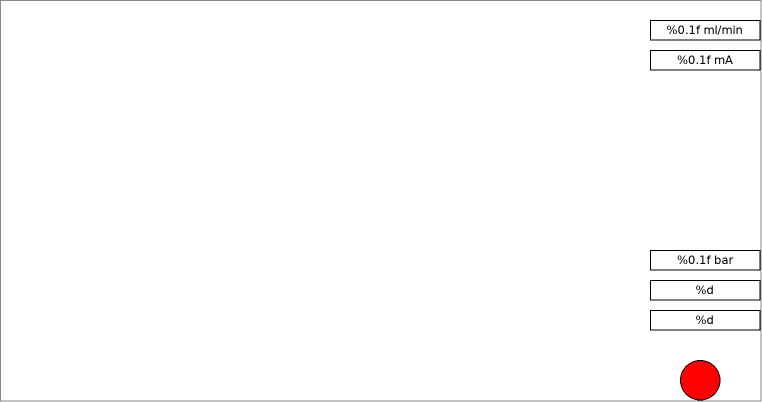
VISUALIZATION Q1  // 762x402
    Rectangle (650,20 110x20), "%0.1f ml/min", text variable: IOs_Variables.Q1_CALCULETED_FLOW
    Rectangle (650,280 110x20), "%d", text variable: LEDS.M1_FB_GetPositionIs.PositionIs
    Rectangle (650,250 110x20), "%0.1f bar", text variable: IOs_Variables.Q1_PRESSURE_SENSOR_VALUE
    Rectangle (650,310 110x20), "%d", text variable: Q1.STEP
    Ellipse (680,360 40x40), colour toggle: (LEDS.M1_FB_GetEnableState.IsEnabled) <> 0
    Rectangle (650,50 110x20), "%0.1f mA", text variable: IOs_Variables.Q1_CURRENT
END_VISUALIZATION

(* stored: Version 1.1.0.1, ProductVersion 3.1.0.26
   Visu Q1: Id {0b9081c7-1e85-4c6a-8c2c-39a2157f4700} *)
